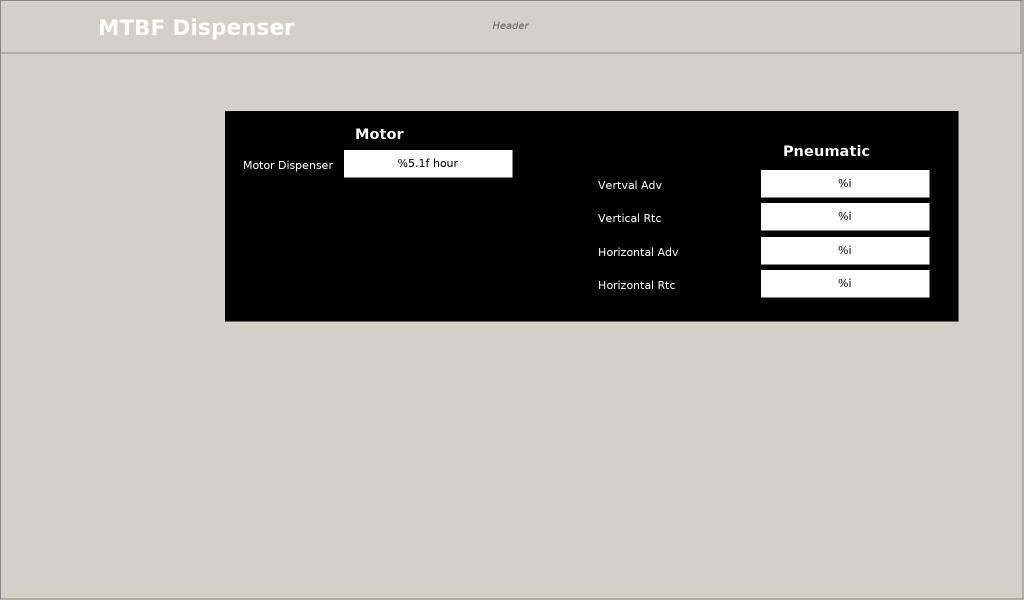
VISUALIZATION MTBF_Dispenser  // 1024x600
    Frame (0,-2 1021x55)
        shows Header()
    Label (95,15 250x25), "MTBF Dispenser"
    RoundedRectangle (225,111 733x210)
    Label (243,114 273x40), "Motor"
    Label (240,148 103x35), "Motor Dispenser"
    RoundedRectangle (343,149 170x29), "%5.1f hour", text variable: InputOutput_GVL.MTBF_Motor[19]
    Label (595,168 147x35), "Vertval Adv"
    RoundedRectangle (760,169 170x29), "%i", text variable: InputOutput_GVL.MTBF_Pneumatic[9]
    Label (690,131 273x40), "Pneumatic"
    Label (595,201 147x35), "Vertical Rtc"
    RoundedRectangle (760,202 170x29), "%i", text variable: InputOutput_GVL.MTBF_Pneumatic[10]
    Label (595,235 147x35), "Horizontal Adv"
    RoundedRectangle (760,236 170x29), "%i", text variable: InputOutput_GVL.MTBF_Pneumatic[11]
    Label (595,268 147x35), "Horizontal Rtc"
    RoundedRectangle (760,269 170x29), "%i", text variable: InputOutput_GVL.MTBF_Pneumatic[12]
END_VISUALIZATION

(* stored: Version 1.1.0.1, ProductVersion 3.1.4024.12
   Visu MTBF_Dispenser: Id {68a2fcec-c496-4824-99bc-68ad8bd8c69c} *)
